(* IEC 61131-3 sources: repolevel_ST_code_completion/dataset/generation_context_ground_truth/barrier, 21 files *)

(* ---- BasePIDCtrl.st ---- *)
VAR
	fCycle			:REAL;
	CycleTime		:TIME ;
	Err				:REAL;    		//本次误差
	LastErr			:REAL;    		//上次误差
	KiErrSum		:REAL;			//积分累计误差
	KdErr			:REAL;			//微分误差
	Result			:REAL;			//计算结果
	Result_OUT		:REAL;		    //限制结果
	trig			:R_TRIG ;
	ton				:TON ;
END_VAR

IF  rCycle < 0.01 THEN  //10ms最小
	fCycle := 0.01;
ELSE
	fCycle := rCycle;
END_IF

CycleTime := REAL_TO_TIME (TIME_TO_REAL(T#1S) * fCycle);
ton (IN := NOT ton.Q ,PT := CycleTime ,Q =>);
trig (CLK := ton.Q  ,Q =>);

IF trig.Q THEN 			//PID计算
	Err := Set_Val - Act_Val;  //误差计算
	KiErrSum := KiErrSum + Err ;   //积分计算
	KdErr := Err -LastErr;    //微分计算
	LastErr := Err;
	(*IF ABS(Err) < 10 THEN		//误差较低时才开启积分
		KiErrSum := KiErrSum + Err ;   //积分计算
	END_IF*)
	Result :=  Kp * Err + Ki * KiErrSum + Kd * KdErr;
END_IF

IF Result > Y_MAX  THEN         //限幅度输出
	Result_OUT := Y_MAX ;
	LimitActive := TRUE ;
ELSIF Result < Y_MIN THEN
	Result_OUT := Y_MIN  ;
	LimitActive := TRUE ;
ELSE
	Result_OUT := Result ;
	LimitActive :=FALSE ;
END_IF
IF Reset THEN   //pid 不输出
	KiErrSum := 0;
	KdErr := 0;
	LastErr	:= 0;
	Y := 0;
ELSE
	Y := Result_OUT;
END_IF

(* ---- CAN_Read_Data_SWMC.st ---- *)
VAR
	frame :Can_baseframe;
END_VAR

CASE  SWMC_ID OF

	1:                       //SWMC-C1
		frame.id 	:= (gCan.C1RxMsg.RXMsg[I].RxMsg_CobId-8)/32;
		frame.data 	:= gCan.C1RxMsg.RXMsg[I].RxMsg_Byte;
	2:                       //SWMC-C2
		frame.id 	:= (gCan.C2RxMsg.RXMsg[I].RxMsg_CobId-8)/32;
		frame.data 	:= gCan.C2RxMsg.RXMsg[I].RxMsg_Byte;
	3:						//SWMC-C3
		frame.id 	:= (gCan.C3RxMsg.RXMsg[I].RxMsg_CobId-8)/32;
		frame.data 	:= gCan.C3RxMsg.RXMsg[I].RxMsg_Byte;
	4:                       //SWMC-C4
		frame.id 	:= (gCan.C4RxMsg.RXMsg[I].RxMsg_CobId-8)/32;
		frame.data 	:= gCan.C4RxMsg.RXMsg[I].RxMsg_Byte;
	//(*
	5:                       //SWMC-C5
		frame.id 	:= (gCan.C5RxMsg.RXMsg[I].RxMsg_CobId-8)/32;
		frame.data 	:= gCan.C5RxMsg.RXMsg[I].RxMsg_Byte;
	6:						//SWMC-C6
		frame.id 	:= (gCan.C6RxMsg.RXMsg[I].RxMsg_CobId-8)/32;
		frame.data 	:= gCan.C6RxMsg.RXMsg[I].RxMsg_Byte;
		//*)
	ELSE				//Other
		frame.id := 0;
		frame.data[1] := 0;
		frame.data[2] := 0;
		frame.data[3] := 0;
		frame.data[4] := 0;
		frame.data[5] := 0;
		frame.data[6] := 0;
		frame.data[7] := 0;
		frame.data[8] := 0;
END_CASE
Can_Read_data_SWMC := frame;

(* ---- CAN_Send_Data_SWMC.st ---- *)
VAR

END_VAR

CASE  SWMC_ID OF

	1:
		gCan.C1TxMsg.TXMsg[1].TxMsg_CobId 	:= 8 + 32 * id;
	  	gCan.C1TxMsg.TXMsg[1].TxMsg_Byte 	:= data;
	   	gCan.C1TxMsg.NoOfTxMessages			:= 1;
	   	gCan.C1TxMsg.TxCounter 				:= gCan.C1TxMsg.TxCounter +1;
	2:
		gCan.C2TxMsg.TXMsg[1].TxMsg_CobId 	:= 8 + 32 * id;
	  	gCan.C2TxMsg.TXMsg[1].TxMsg_Byte 	:= data;
	   	gCan.C2TxMsg.NoOfTxMessages			:= 1;
	   	gCan.C2TxMsg.TxCounter 				:= gCan.C2TxMsg.TxCounter +1;
	3:
		gCan.C3TxMsg.TXMsg[1].TxMsg_CobId 	:= 8 + 32 * id;
	  	gCan.C3TxMsg.TXMsg[1].TxMsg_Byte 	:= data;
	   	gCan.C3TxMsg.NoOfTxMessages			:= 1;
	   	gCan.C3TxMsg.TxCounter 				:= gCan.C3TxMsg.TxCounter +1;
	4:
		gCan.C4TxMsg.TXMsg[1].TxMsg_CobId 	:= 8 + 32 * id;
	  	gCan.C4TxMsg.TXMsg[1].TxMsg_Byte 	:= data;
	   	gCan.C4TxMsg.NoOfTxMessages			:= 1;
	   	gCan.C4TxMsg.TxCounter 				:= gCan.C4TxMsg.TxCounter +1;
	//(*
	5:
		gCan.C5TxMsg.TXMsg[1].TxMsg_CobId 	:= 8 + 32 * id;
	  	gCan.C5TxMsg.TXMsg[1].TxMsg_Byte 	:= data;
	   	gCan.C5TxMsg.NoOfTxMessages			:= 1;
	   	gCan.C5TxMsg.TxCounter 				:= gCan.C5TxMsg.TxCounter +1;
	6:
		gCan.C6TxMsg.TXMsg[1].TxMsg_CobId 	:= 8 + 32 * id;
	  	gCan.C6TxMsg.TXMsg[1].TxMsg_Byte 	:= data;
	   	gCan.C6TxMsg.NoOfTxMessages			:= 1;
	   	gCan.C6TxMsg.TxCounter 				:= gCan.C6TxMsg.TxCounter +1;
	//*)

END_CASE

(* ---- CommandExecutor.st ---- *)
VAR
END_VAR

IF percent > 0 THEN
	CASE level OF
		1:
			gController.grd[idx].extendPercent := REAL_TO_WORD(percent * 65535 / 100);
			gController.grd[idx].retractPercent := 0;
		2:
			gController.sky[idx].extendPercent := REAL_TO_WORD(percent * 65535 / 100);
			gController.sky[idx].retractPercent := 0;
	END_CASE
ELSE
	CASE level OF
		1:
			gController.grd[idx].extendPercent := 0;
			gController.grd[idx].retractPercent := REAL_TO_WORD(ABS(percent) * 65535 / 100);
		2:
			gController.sky[idx].extendPercent := 0;
			gController.sky[idx].retractPercent := REAL_TO_WORD(ABS(percent) * 65535 / 100);
	END_CASE
END_IF

(* ---- CommandExecutor0.st ---- *)
VAR
END_VAR

CASE direct OF
	TargetDirect.extend:
		CASE level OF
			1:
				gController.grd[idx].extendPercent := REAL_TO_WORD(percent * 65535 / 100);
				gController.grd[idx].retractPercent := 0;
			2:
				gController.sky[idx].extendPercent := REAL_TO_WORD(percent * 65535 / 100);
				gController.sky[idx].retractPercent := 0;
		END_CASE
	TargetDirect.retract:
		CASE level OF
			1:
				gController.grd[idx].extendPercent := 0;
				gController.grd[idx].retractPercent := REAL_TO_WORD(percent * 65535 / 100);
			2:
				gController.sky[idx].extendPercent := 0;
				gController.sky[idx].retractPercent := REAL_TO_WORD(percent * 65535 / 100);
		END_CASE
	TargetDirect.stop:
		CASE level OF
			1:
				gController.grd[idx].extendPercent := 0;
				gController.grd[idx].retractPercent := 0;
			2:
				gController.sky[idx].extendPercent := 0;
				gController.sky[idx].retractPercent := 0;
		END_CASE

	ELSE
		CASE level OF
			1:
				gController.grd[idx].extendPercent := 0;
				gController.grd[idx].retractPercent := 0;
			2:
				gController.sky[idx].extendPercent := 0;
				gController.sky[idx].retractPercent := 0;
		END_CASE

END_CASE

(* ---- DataReverse.st ---- *)
VAR
END_VAR

(* ---- DataReverse_cmdReverse.st ---- *)
IF input = TargetDirect.extend THEN
	cmdReverse := TargetDirect.retract;
END_IF
IF input = TargetDirect.retract THEN
	cmdReverse := TargetDirect.extend;
END_IF

(* ---- fileSave.st ---- *)
VAR
	lineCount	: INT;
	fileHandle  : DWORD;
	fileName	: STRING;
END_VAR
VAR_OUTPUT
END_VAR

(* ---- fileSave_close.st ---- *)
VAR
	lineCount	: INT;
	fileHandle  : DWORD;
	fileName	: STRING;
END_VAR
VAR_OUTPUT
END_VAR

IF fileHandle <> 0 THEN
	SysFileClose(hFile := fileHandle);
	fileHandle := 0;
END_IF

(* ---- fileSave_createDir.st ---- *)
VAR
	lineCount	: INT;
	fileHandle  : DWORD;
	fileName	: STRING;
	filePath1	:STRING;
END_VAR
VAR_OUTPUT
END_VAR

filePath1 := FilePath;
filePath1 := concat(filePath1,'/');
filePath1 := concat(filePath1,devName);
SysDirCreate2(filePath1, TRUE);

(* ---- fileSave_new.st ---- *)
VAR
	lineCount	: INT;
	fileHandle  : DWORD;
	fileName	: STRING;
	fileHandle0 : DWORD;
	datetime	: DATE_AND_TIME;
	UdIntms 	: UDINT;
	UdMsOffset  : UDINT;
	DTimer_Str  : STRING;
	uiYear 		: UINT;
    uiMonth 	: UINT;
    uiDay 		: UINT;
    uiHour 		: UINT;
    uiMinute 	: UINT;
    uiSecond 	: UINT;
	uiMsSecond	: UINT;

	S_Time64		:  SysTime64;
	STT			:  CurTimeEx;
	S_Time			:  SystemTimeDate;
	Time_Str		:  STRING;
	F_err		: DWORD;
	F_HANDL		: DWORD;
END_VAR
VAR_OUTPUT
END_VAR

	STT(SystemTime:= S_Time64, TimeDate:= S_Time);
	Time_Str :='';
	Time_Str := concat(Time_Str,UINT_TO_STRING(S_Time.Year));
	Time_Str := concat(Time_Str,'-');
	Time_Str := concat(Time_Str,UINT_TO_STRING(S_Time.Month));
	Time_Str := concat(Time_Str,'-');
	Time_Str := concat(Time_Str,UINT_TO_STRING(S_Time.Day));
	Time_Str := concat(Time_Str,'_');
	Time_Str := concat(Time_Str,UINT_TO_STRING(S_Time.Hour));
	Time_Str := concat(Time_Str,'-');
	Time_Str := concat(Time_Str,UINT_TO_STRING(S_Time.Minute));
	Time_Str := concat(Time_Str,'-');
	Time_Str := concat(Time_Str,UINT_TO_STRING(S_Time.Second));
	Time_Str := concat(Time_Str,'_');
	Time_Str := concat(Time_Str,UINT_TO_STRING(S_Time.Milliseconds));

	fileName := FilePath;
	fileName := concat(fileName,'/');
	fileName := concat(fileName,devName);

	fileName := concat(fileName,'/');
	fileName := concat(fileName,devName);
	fileName := concat(fileName,'-');
	fileName := concat(fileName,Time_Str);
    fileName := concat(fileName,'.txt');

	fileHandle := SysFileOpen(szFile:= fileName, am:=ACCESS_MODE.AM_WRITE, pResult:= ADR(F_err));
	lineCount := -1;
	//fileHandle := SysFileOpen(szFile:= fileName, am:=ACCESS_MODE.AM_APPEND, pResult:= ADR(F_err));

(* ---- fileSave_write.st ---- *)
VAR
	lineCount	: INT;
	fileHandle  : DWORD;
	fileName	: STRING;
	data		: STRING;
	F_err		: DWORD;
	tempInt		: INT;
END_VAR
VAR_OUTPUT
END_VAR

IF fileHandle <> 0 THEN
	lineCount := lineCount + 1;
	tempInt	:= lineCount * intervalt;
	data := INT_TO_STRING(lineCount);
	data := concat(data,'$T$T');
	data := concat(data, INT_TO_STRING(tempInt));
	IF tempInt < 1000 THEN
		data := concat(data,'$T');
	END_IF
	data := concat(data,'$T$T');
	data := concat(data,INT_TO_STRING(positionInt));
	data := concat(data,'$T');
	data := concat(data,INT_TO_STRING(speedInt));
	data := concat(data,'$T');
	data := concat(data,INT_TO_STRING(stateInt));
	data := concat(data,'$R');

	SysFileWrite(hFile:=fileHandle , pbyBuffer:= ADR(data) , ulSize:= DINT_TO_DWORD(SysStrLen(data)) , pResult:= ADR(F_err));		// 写入数据

END_IF

(* ---- grdPosCtrl.st ---- *)
VAR
	posPid		:BasePIDCtrl;
	spdPid		:BasePIDCtrl;
	setSpeed	:REAL;
	overBase	:REAL;
	out			:REAL;
	controller	:DevPid;
END_VAR

controller := gDev.grd[idx].ctrl;
posPid(
	Act_Val:= gDev.grd[idx].sensor.position,
	Set_Val:= controller.pos.Set_Point,
	Kp:= controller.pos.Kp,
	Ki:= controller.pos.Ki,
	Kd:= controller.pos.Kd,
	Y_MAX:= controller.pos.Max_Val,     //最大速度
	Y_MIN:= -controller.pos.Max_Val,    //水平运动正反一致
	rCycle:= 0.1,   //位置计算周期 100ms
	Reset:= isReset,
	Y => controller.pos.OUT,
	LimitActive=> );

IF ABS(posPid.Y - setSpeed) > (cycTimer * controller.pos.Max_ACC) THEN
	IF posPid.Y > setSpeed THEN
		setSpeed := setSpeed + (cycTimer * controller.pos.Max_ACC);
	ELSE
		setSpeed := setSpeed - (cycTimer * controller.pos.Max_ACC);
	END_IF
ELSE
	setSpeed := posPid.Y;
END_IF

controller.spd.Set_Point := setSpeed;

IF setSpeed > 0 THEN
	overBase := setSpeed * controller.ff.pstKv + controller.ff.pstThreshold;
ELSE
	overBase := setSpeed * controller.ff.negKv - controller.ff.negThreshold;
END_IF

spdPid(
	Act_Val:= gDev.grd[idx].sensor.speed,
	Set_Val:= controller.spd.Set_Point,
	Kp:= controller.spd.Kp,
	Ki:= controller.spd.Ki,
	Kd:= controller.spd.Kd,
	Y_MAX:= controller.spd.Max_Val,     //最大速度
	Y_MIN:= -controller.spd.Max_Val,    //水平运动正反一致
	rCycle:= 0.02,   //位置计算周期 100ms
	Reset:= isReset,
	Y=> ,
	LimitActive=> );

out := spdPid.Y + overBase;
IF out > controller.spd.Max_Val THEN
	out := controller.spd.Max_Val;
END_IF
IF out < -controller.spd.Max_Val THEN
	out := -controller.spd.Max_Val;
END_IF
IF isReset	THEN out := 0;	END_IF
controller.spd.OUT := out;
gDev.grd[idx].ctrl := controller;
res := out;

(* ---- mdbsLogicToPhy.st ---- *)
VAR
END_VAR

(**
 * 将华中指令解析为要动作挡板的标号
 * (level:1->地轨	2->天轨)(phyIdx:内存物理地址对应数组索引)
 *)
CASE section OF
	1://区域限定1:skyExtend)
		level := 2;
		direct := TargetDirect.extend;
		CASE lgcIdx OF
			1:	phyIdx := 1;		//横1	->	sky1
			2:	phyIdx := 3;		//横2	->	sky3
			3:	phyIdx := 4;		//横3	->	sky4
			4:	phyIdx := 5;		//横4	->	sky5
			5:	phyIdx := 6;		//横5	->	sky6
			6:	phyIdx := 8;		//横6	->	sky8
			7:	phyIdx := 9;		//横7	->	sky9
			8:	phyIdx := 10;		//横8	->	sky10
			9:	phyIdx := 2;		//纵1	->	sky2
			10:	phyIdx := 7;		//纵2	->	sky7
			11:	phyIdx := 0;		//起竖	->	sky0
		END_CASE

	2://区域限定2:skyRetract)
		level := 2;
		direct := TargetDirect.retract;
		CASE lgcIdx OF
			1:	phyIdx := 1;		//横1	->	sky1
			2:	phyIdx := 3;		//横2	->	sky3
			3:	phyIdx := 4;		//横3	->	sky4
			4:	phyIdx := 5;		//横4	->	sky5
			5:	phyIdx := 6;		//横5	->	sky6
			6:	phyIdx := 8;		//横6	->	sky8
			7:	phyIdx := 9;		//横7	->	sky9
			8:	phyIdx := 10;		//横8	->	sky10
			9:	phyIdx := 2;		//纵1	->	sky2
			10:	phyIdx := 7;		//纵2	->	sky7
			11:	phyIdx := 0;		//起竖	->	sky0
		END_CASE

	3://区域限定3:grdExtend)
		level := 1;
		direct := TargetDirect.extend;
		CASE lgcIdx OF
			1:	phyIdx := 1;		//横1	->	grd1
			2:	phyIdx := 3;		//横2	->	grd3
			3:	phyIdx := 4;		//横3	->	grd4
			4:	phyIdx := 5;		//横4	->	grd5
			5:	phyIdx := 6;		//横5	->	grd6
			6:	phyIdx := 8;		//横6	->	grd8
			7:	phyIdx := 9;		//横7	->	grd9
			8:	phyIdx := 10;		//横8	->	grd10
			9:	phyIdx := 2;		//纵1	->	grd2
			10:	phyIdx := 7;		//纵2	->	grd7
		END_CASE
	4://区域限定4:grdRetract)
		level := 1;
		direct := TargetDirect.retract;
		CASE lgcIdx OF
			1:	phyIdx := 1;
			2:	phyIdx := 3;
			3:	phyIdx := 4;
			4:	phyIdx := 5;
			5:	phyIdx := 6;
			6:	phyIdx := 8;
			7:	phyIdx := 9;
			8:	phyIdx := 10;
			9:	phyIdx := 2;
			10:	phyIdx := 7;
		END_CASE
END_CASE

(* ---- mdbsNumToIdx.st ---- *)
VAR

END_VAR

IF devNo > 40000 THEN
	CASE devNo OF
		//地轨
		41010:	level := 1;	idx := 1;
		41020:	level := 1;	idx := 3;
		41030:	level := 1;	idx := 4;
		41040:	level := 1;	idx := 5;
		41050:	level := 1;	idx := 6;
		41060:	level := 1;	idx := 8;
		41070:	level := 1;	idx := 9;
		41080:	level := 1;	idx := 10;
		42010:	level := 1;	idx := 2;
		42020:	level := 1;	idx := 7;

		51010:	level := 2;	idx := 1;
		51020:	level := 2;	idx := 3;
		51030:	level := 2;	idx := 4;
		51040:	level := 2;	idx := 5;
		51050:	level := 2;	idx := 6;
		51060:	level := 2;	idx := 8;
		51070:	level := 2;	idx := 9;
		51080:	level := 2;	idx := 10;
		52010:	level := 2;	idx := 2;
		52020:	level := 2;	idx := 7;
		53000:	level := 2;	idx := 0;
		53010:	level := 2;	idx := 0;
	END_CASE
END_IF

(* ---- mdbsPhyToLogic.st ---- *)
VAR
END_VAR

(**
 * 输入挡板标号，返回华中需要的寄存器地址号
 *)
CASE section OF
	1://区域限定(1:groundExtend)
		CASE phyIdx OF
			1:	lgcIdx := 223;		//grd1e	->	横1	223
			2:	lgcIdx := 231;		//grd2e	->	纵1	231
			3:	lgcIdx := 224;		//grd3e	->	横2	224
			4:	lgcIdx := 225;		//grd4e	->	横3	225
			5:	lgcIdx := 226;		//grd5e	->	横4	226
			6:	lgcIdx := 227;		//grd6e	->	横5	227
			7:	lgcIdx := 232;		//grd7e	->	纵2	232
			8:	lgcIdx := 228;		//grd8e	->	横6	228
			9:	lgcIdx := 229;		//grd9e	->	横7	229
			10:	lgcIdx := 230;		//grd10e->	横8	230
		END_CASE
	2://区域限定(2:groundRetract)
		CASE phyIdx OF
			1:	lgcIdx := 271;		//grd1r	->	横1
			2:	lgcIdx := 279;		//grd2r	->	纵1
			3:	lgcIdx := 272;		//grd3r	->	横2
			4:	lgcIdx := 273;		//grd4r	->	横3
			5:	lgcIdx := 274;		//grd5r	->	横4
			6:	lgcIdx := 275;		//grd6r	->	横5
			7:	lgcIdx := 280;		//grd7r	->	纵2
			8:	lgcIdx := 276;		//grd8r	->	横6
			9:	lgcIdx := 277;		//grd9r	->	横7
			10:	lgcIdx := 278;		//grd10r->	横8
		END_CASE
	3://区域限定(3:skyExtend)
		CASE phyIdx OF
			0:	lgcIdx := 137;		//sky0e	->	起竖
			1:	lgcIdx := 127;		//sky1e	->	横1
			2:	lgcIdx := 135;		//sky2e	->	纵1
			3:	lgcIdx := 128;		//sky3e	->	横2
			4:	lgcIdx := 129;		//sky4e	->	横3
			5:	lgcIdx := 130;		//sky5e	->	横4
			6:	lgcIdx := 131;		//sky6e	->	横5
			7:	lgcIdx := 136;		//sky7e	->	纵2
			8:	lgcIdx := 132;		//sky8e	->	横6
			9:	lgcIdx := 133;		//sky9e	->	横7
			10:	lgcIdx := 134;		//sky10e->	横8
		END_CASE

	4://区域限定(4:skyRetract)
		CASE phyIdx OF
			0:	lgcIdx := 185;		//sky0r	->	起竖
			1:	lgcIdx := 175;		//sky1r	->	横1
			2:	lgcIdx := 183;		//sky2r	->	纵1
			3:	lgcIdx := 176;		//sky3r	->	横2
			4:	lgcIdx := 177;		//sky4r	->	横3
			5:	lgcIdx := 178;		//sky5r	->	横4
			6:	lgcIdx := 179;		//sky6r	->	横5
			7:	lgcIdx := 184;		//sky7r	->	纵2
			8:	lgcIdx := 180;		//sky8r	->	横6
			9:	lgcIdx := 181;		//sky9r	->	横7
			10:	lgcIdx := 182;		//sky10r->	横8
		END_CASE
END_CASE

(* ---- percentCalc.st ---- *)
VAR
	c			:REAL;
	p			:REAL;
END_VAR

//伸出百分比计算
CASE level OF
	1:
		IF gDev.grd[idx].sensor.position < 3 THEN
			RETURN;
		END_IF
		c := gDev.grd[idx].sensor.position - gDev.grd[idx].sensor.retractVal;
		p := gDev.grd[idx].sensor.extendVal - gDev.grd[idx].sensor.retractVal;
		percentCalc := c * 100 / p;
	2:
		IF gDev.sky[idx].sensor.position < 3 THEN
			RETURN;
		END_IF
		c := gDev.sky[idx].sensor.position - gDev.sky[idx].sensor.retractVal;
		p := gDev.sky[idx].sensor.extendVal - gDev.sky[idx].sensor.retractVal;
		percentCalc := c * 100 / p;
END_CASE

(* ---- setButtonByDirect.st ---- *)
VAR
END_VAR
//	本函数用于根据输入参数 操作UI界面的按钮变量
CASE level OF
	1:
		IF idx = 0 OR idx > 10 THEN		//参数校验
			RETURN;
		END_IF
		CASE direct OF
			TargetDirect.extend:
				gUI.grd[idx].btnStop := FALSE;
				gUI.grd[idx].btnExtend := TRUE;
				gUI.grd[idx].btnRetract := FALSE;
			TargetDirect.retract:
				gUI.grd[idx].btnStop := FALSE;
				gUI.grd[idx].btnExtend := FALSE;
				gUI.grd[idx].btnRetract := TRUE;
			TargetDirect.stop:
				gUI.grd[idx].btnStop := FALSE;
				gUI.grd[idx].btnExtend := FALSE;
				gUI.grd[idx].btnRetract := FALSE;
		END_CASE
	2:
		IF idx > 10 THEN		//参数校验
			RETURN;
		END_IF
		CASE direct OF
			TargetDirect.extend:
				gUI.sky[idx].btnStop := FALSE;
				gUI.sky[idx].btnExtend := TRUE;
				gUI.sky[idx].btnRetract := FALSE;
			TargetDirect.retract:
				gUI.sky[idx].btnStop := FALSE;
				gUI.sky[idx].btnExtend := FALSE;
				gUI.sky[idx].btnRetract := TRUE;
			TargetDirect.stop:
				gUI.sky[idx].btnStop := FALSE;
				gUI.sky[idx].btnExtend := FALSE;
				gUI.sky[idx].btnRetract := FALSE;
		END_CASE

END_CASE;

(* ---- skyPosCtrl.st ---- *)
VAR
	posPid		:BasePIDCtrl;
	spdPid		:BasePIDCtrl;
	setSpeed	:REAL;
	overBase	:REAL;
	out			:REAL;
	//fb_Val		:REAL;
	controller	:DevPid;
END_VAR

controller := gDev.sky[idx].ctrl;
posPid(
	Act_Val:= gDev.sky[idx].sensor.position,
	Set_Val:= controller.pos.Set_Point,
	Kp:= controller.pos.Kp,
	Ki:= controller.pos.Ki,
	Kd:= controller.pos.Kd,
	Y_MAX:= controller.pos.Max_Val,     //最大速度
	Y_MIN:= -controller.pos.Max_Val,    //水平运动正反一致
	rCycle:= 0.05,   //位置计算周期 100ms
	Reset:= isReset,
	Y => controller.pos.OUT,
	LimitActive=> );

IF ABS(posPid.Y - setSpeed) > (cycTimer * controller.pos.Max_ACC) THEN
	IF posPid.Y > setSpeed THEN
		setSpeed := setSpeed + (cycTimer * controller.pos.Max_ACC);
	ELSE
		setSpeed := setSpeed - (cycTimer * controller.pos.Max_ACC);
	END_IF
ELSE
	setSpeed := posPid.Y;
END_IF

controller.spd.Set_Point := setSpeed;

IF setSpeed > 0 THEN
	overBase := setSpeed * controller.ff.pstKv + controller.ff.pstThreshold;
END_IF
IF setSpeed < 0 THEN
	overBase := setSpeed * controller.ff.negKv - controller.ff.negThreshold;
END_IF

spdPid(
	Act_Val:= gDev.sky[idx].sensor.speed,
	Set_Val:= controller.spd.Set_Point,
	Kp:= controller.spd.Kp,
	Ki:= controller.spd.Ki,
	Kd:= controller.spd.Kd,
	Y_MAX:= controller.spd.Max_Val,     //最大速度
	Y_MIN:= -controller.spd.Max_Val,    //水平运动正反一致
	rCycle:= 0.02,   //位置计算周期 100ms
	Reset:= isReset,
	Y=> ,
	LimitActive=> );

out := spdPid.Y + overBase;

IF out > controller.spd.Max_Val THEN
	out := controller.spd.Max_Val;
END_IF
IF out < -controller.spd.Max_Val THEN
	out := -controller.spd.Max_Val;
END_IF
IF isReset	THEN out := 0;	END_IF
controller.spd.OUT := out;
gDev.sky[idx].ctrl := controller;
res := out;

(* ---- tcpUpload_send.st ---- *)
VAR
	tcpConnector	:TCP.Connector;
	tcpStream		:TCP.Stream;
	pointerStream	:POINTER TO TCP.Stream;
	sizeData		:__XINT;

	tcpState		:UINT:=0;
	tcpCount		:UINT:=0;

	netState		:INT;
END_VAR

tcpCount := tcpCount + 1;
CASE tcpState OF

	0:			//connet server
		tcpConnector.Connect(sIPAddress:= InetAddress,uiPort:= port,pStream => pointerStream);
		IF pointerStream<>0 THEN
			tcpState :=1;
		ELSE
			tcpState :=2;
		END_IF

	1:
		netState := pointerStream^.Send(ADR(sendBuf),dataLength,diSent=>sizeData);
		IF netState <> 0 THEN
			tcpState := 2;
		END_IF

	2:		 	//断开连接
	    tcpConnector.Disconnect();
		tcpState := 0;

END_CASE

(* ---- updateDevStatus.st ---- *)
VAR
	extendVal	:REAL;		//伸出值
	retractVal	:REAL;		//缩回到位值
	nowVal		:REAL;		//当前值
	stat		:DevStatus;	//设备状态
END_VAR

(* 本函数用于根据设备的标定伸出/缩回值以及当前位置
** 判断该缸体是否处于伸出/缩回到位状态，如果到位更新参数
*)

stat := DevStatus.unknown;	//初始化状态量
CASE level OF
	1:
		extendVal := gDev.grd[idx].sensor.extendVal;
		retractVal := gDev.grd[idx].sensor.retractVal;
		nowVal := gDev.grd[idx].sensor.position;
		stat := gDev.grd[idx].state;
	2:
		extendVal := gDev.sky[idx].sensor.extendVal;
		retractVal := gDev.sky[idx].sensor.retractVal;
		nowVal := gDev.sky[idx].sensor.position;
		stat := gDev.sky[idx].state;
END_CASE

IF nowVal > 1 THEN
	IF nowVal < retractVal + errorVal THEN
		stat := DevStatus.retracted;
	ELSIF nowVal > extendVal - errorVal THEN
		stat := DevStatus.extended;
	ELSE
		IF stat <> DevStatus.runing THEN
			stat := DevStatus.error;
		END_IF
	END_IF
ELSE
	stat := DevStatus.unknown;
END_IF

CASE level OF
	1:
		gDev.grd[idx].state := stat;
	2:
		gDev.sky[idx].state := stat;
END_CASE

updateDevStatus := stat;
